FUNCTION_BLOCK FB_ObserverPattern_Test EXTENDS TcUnit.FB_TestSuite
// All observable types implements the same base methods for
// managing the list of observers, hence testing only one type
// of observable is enough. For instance, methods like, `Attach`,
// and `Detach`.
VAR
    fVal: LREAL;
END_VAR

TestAdd5CompatibleObserversExpectAll5();
TestAdd6IncompatibleObserversExpectNone();
TestAddDuplicateObserversExpectFailure();
TestAddMoreObserversThanAllowedExpectOnlyMaxCount();
TestCompatibleDataTypesExpectValuesToUpdate();
TestDataTypeConsistencyOfObservables();
TestDataTypeConsistencyOfObservers();
TestDetachAddedObserversExpectSuccess();
TestIncompatileDataTypesExpectNoValueChange();
TestObservableNotifyAlwaysUponWriteAccess();
TestObservableNotifyOnlyWhenValueChanged();
TestObservableNotifyUponAttachmentWithObservers();
TestObserverExternalWithCompatibleDataTypeExpectValueToUpdate();
TestOneObservableToManyObserversExpectAllToUpdateValueAccordingly();

METHOD PRIVATE TestAdd5CompatibleObserversExpectAll5
VAR_INST
    fbObservableReal: FB_Observable_REAL(TRUE);

    aObserverReal: ARRAY [1..5] OF FB_Observer_REAL;

    i: UDINT;
END_VAR
TcUnit.TEST('TestAdd5CompatibleObserversExpectAll5');

FOR i := 1 TO SIZEOF(aObserverReal)/SIZEOF(aObserverReal[1]) DO
    THIS^.AssertTrue(Condition := fbObservableReal.Attach(aObserverReal[i]),
                     Message := 'Failed to add compatible observer to observable');
END_FOR

THIS^.AssertEquals_UDINT(Expected := 5,
                         Actual := fbObservableReal.nObserverCount,
                         Message := 'Unexpected number of observers attached');

TcUnit.TEST_FINISHED();
END_METHOD

METHOD PRIVATE TestAdd6IncompatibleObserversExpectNone
VAR_INST
    // Test can be less manual with dynamic list
    fbObservableDint: FB_Observable_DINT(TRUE);
    fbObservableUdint: FB_Observable_UDINT(TRUE);
    fbObservableUint: FB_Observable_UINT(TRUE);
    fbObservableReal: FB_Observable_REAL(TRUE);
    fbObservableLreal: FB_Observable_LREAL(TRUE);

    fbObserverDint: ARRAY [1..6] OF FB_Observer_DINT;
    fbObserverUdint: ARRAY [1..6] OF FB_Observer_UDINT;
    fbObserverUint: ARRAY [1..6] OF FB_Observer_UINT;
    fbObserverLreal: ARRAY [1..6] OF FB_Observer_LREAL;
    fbObserverReal: ARRAY [1..6] OF FB_Observer_REAL;

    i: UDINT;
END_VAR
TcUnit.TEST('TestAdd6IncompatibleObserversExpectNone');

FOR i := 1 TO SIZEOF(fbObserverUdint)/SIZEOF(fbObserverUdint[1]) DO
    fbObservableDint.Attach(fbObserverUdint[i]);
    fbObservableDint.Attach(fbObserverUint[i]);
    fbObservableDint.Attach(fbObserverLreal[i]);
    fbObservableDint.Attach(fbObserverReal[i]);

    fbObservableUdint.Attach(fbObserverDint[i]);
    fbObservableUdint.Attach(fbObserverUint[i]);
    fbObservableUdint.Attach(fbObserverLreal[i]);
    fbObservableUdint.Attach(fbObserverReal[i]);

    fbObservableUint.Attach(fbObserverDint[i]);
    fbObservableUint.Attach(fbObserverUdint[i]);
    fbObservableUint.Attach(fbObserverLreal[i]);
    fbObservableUint.Attach(fbObserverReal[i]);

    fbObservableLreal.Attach(fbObserverDint[i]);
    fbObservableLreal.Attach(fbObserverUdint[i]);
    fbObservableLreal.Attach(fbObserverUint[i]);
    fbObservableLreal.Attach(fbObserverReal[i]);

    fbObservableReal.Attach(fbObserverDint[i]);
    fbObservableReal.Attach(fbObserverUdint[i]);
    fbObservableReal.Attach(fbObserverUint[i]);
    fbObservableReal.Attach(fbObserverLreal[i]);

END_FOR

THIS^.AssertEquals_UDINT(Expected := 0,
                         Actual := fbObservableDint.nObserverCount,
                         Message := 'Unexpected number of observers attached to observable type DINT');

THIS^.AssertEquals_UDINT(Expected := 0,
                         Actual := fbObservableUdint.nObserverCount,
                         Message := 'Unexpected number of observers attached to observable type UDINT');

THIS^.AssertEquals_UDINT(Expected := 0,
                         Actual := fbObservableUint.nObserverCount,
                         Message := 'Unexpected number of observers attached to observable type UINT');

THIS^.AssertEquals_UDINT(Expected := 0,
                         Actual := fbObservableLreal.nObserverCount,
                         Message := 'Unexpected number of observers attached to observable type LREAL');

THIS^.AssertEquals_UDINT(Expected := 0,
                         Actual := fbObservableReal.nObserverCount,
                         Message := 'Unexpected number of observers attached to observable type REAL');

TcUnit.TEST_FINISHED();
END_METHOD

METHOD PRIVATE TestAddDuplicateObserversExpectFailure
VAR_INST
    fbObservableReal: FB_Observable_REAL(TRUE);

    fbObserverReal: FB_Observer_REAL;

    i: UDINT;
END_VAR
TcUnit.TEST('TestAddDuplicateObserversExpectFailure');

FOR i := 1 TO 5 DO
    IF i = 1 THEN
        THIS^.AssertTrue(Condition := fbObservableReal.Attach(fbObserverReal),
                         Message := 'Failed to add compatible observer to observable');
    ELSE
        THIS^.AssertFalse(Condition := fbObservableReal.Attach(fbObserverReal),
                          Message := 'Observable should not add duplicate observers');
    END_IF
END_FOR

THIS^.AssertEquals_UDINT(Expected := 1,
                         Actual := fbObservableReal.nObserverCount,
                         Message := 'Unexpected number of observers attached');

TcUnit.TEST_FINISHED();
END_METHOD

METHOD PRIVATE TestAddMoreObserversThanAllowedExpectOnlyMaxCount
VAR_INST
    fbObservableReal: FB_Observable_REAL(TRUE);

    fbObserverReal: ARRAY [1..(TcBase.Param_Observer.cMaxNumberOfObservers+10)] OF FB_Observer_REAL;

    i: UDINT;
END_VAR
TcUnit.TEST('TestAddMoreObserversThanAllowedExpectOnlyMaxCount');

FOR i := 1 TO SIZEOF(fbObserverReal)/SIZEOF(fbObserverReal[1]) DO
    fbObservableReal.Attach(fbObserverReal[i]);
END_FOR

THIS^.AssertEquals_UDINT(Expected := TcBase.Param_Observer.cMaxNumberOfObservers,
                         Actual := fbObservableReal.nObserverCount,
                         Message := 'Unexpected number of observers attached');

TcUnit.TEST_FINISHED();
END_METHOD

METHOD PRIVATE TestCompatibleDataTypesExpectValuesToUpdate
VAR_INST
    fbObservableBool: FB_Observable_BOOL(TRUE);
    fbObservableByte: FB_Observable_BYTE(TRUE);
    fbObservableWord: FB_Observable_WORD(TRUE);
    fbObservableDword: FB_Observable_DWORD(TRUE);
    fbObservableLword: FB_Observable_LWORD(TRUE);
    fbObservableSint: FB_Observable_SINT(TRUE);
    fbObservableUsint: FB_Observable_USINT(TRUE);
    fbObservableInt: FB_Observable_INT(TRUE);
    fbObservableUint: FB_Observable_UINT(TRUE);
    fbObservableDint: FB_Observable_DINT(TRUE);
    fbObservableUdint: FB_Observable_UDINT(TRUE);
    fbObservableLint: FB_Observable_LINT(TRUE);
    fbObservableUlint: FB_Observable_ULINT(TRUE);
    fbObservableLreal: FB_Observable_LREAL(TRUE);
    fbObservableReal: FB_Observable_REAL(TRUE);

    fbObserverBool: FB_Observer_BOOL;
    fbObserverByte: FB_Observer_BYTE;
    fbObserverWord: FB_Observer_WORD;
    fbObserverDword: FB_Observer_DWORD;
    fbObserverLword: FB_Observer_LWORD;
    fbObserverSint: FB_Observer_SINT;
    fbObserverUsint: FB_Observer_USINT;
    fbObserverInt: FB_Observer_INT;
    fbObserverUint: FB_Observer_UINT;
    fbObserverDint: FB_Observer_DINT;
    fbObserverUdint: FB_Observer_UDINT;
    fbObserverLint: FB_Observer_LINT;
    fbObserverUlint: FB_Observer_ULINT;
    fbObserverLreal: FB_Observer_LREAL;
    fbObserverReal: FB_Observer_REAL;

    bVal: BOOL;
    i: UDINT;
END_VAR
TcUnit.TEST('TestCompatibleDataTypesExpectValuesToUpdate');

fbObservableBool.Attach(fbObserverBool);
fbObservableByte.Attach(fbObserverByte);
fbObservableWord.Attach(fbObserverWord);
fbObservableDword.Attach(fbObserverDword);
fbObservableLword.Attach(fbObserverLword);
fbObservableSint.Attach(fbObserverSint);
fbObservableUsint.Attach(fbObserverUsint);
fbObservableUint.Attach(fbObserverUint);
fbObservableInt.Attach(fbObserverInt);
fbObservableDint.Attach(fbObserverDint);
fbObservableUdint.Attach(fbObserverUdint);
fbObservableLint.Attach(fbObserverLint);
fbObservableUlint.Attach(fbObserverUlint);
fbObservableLreal.Attach(fbObserverLreal);
fbObservableReal.Attach(fbObserverReal);

FOR i := 1 TO 10 DO
    bVal := NOT bVal;
    fbObservableBool.bVal := bVal;
    fbObservableByte.nValue8 := TO_BYTE(i);
    fbObservableWord.nValue16 := TO_WORD(i);
    fbObservableDword.nValue32 := TO_DWORD(i);
    fbObservableLword.nValue64 := TO_LWORD(i);
    fbObservableSint.nValue8 := TO_SINT(i);
    fbObservableUsint.nValue8 := TO_USINT(i);
    fbObservableInt.nValue16 := TO_INT(i);
    fbObservableUint.nValue16 := TO_UINT(i);
    fbObservableDint.nValue32 := TO_DINT(i);
    fbObservableUdint.nValue32 := i;
    fbObservableLint.nValue64 := TO_LINT(i);
    fbObservableUlint.nValue64 := TO_ULINT(i);
    fbObservableLreal.fValue64 := TO_LREAL(i);
    fbObservableReal.fValue32 := TO_REAL(i);

    THIS^.AssertEquals_BOOL(Expected := bVal,
                            Actual := fbObserverBool.bValue,
                            Message := 'BOOL observer failed to update value according to observable');
    THIS^.AssertEquals_BYTE(Expected := TO_BYTE(i),
                            Actual := fbObserverByte.nValue8,
                            Message := 'BYTE observer failed to update value according to observable');
    THIS^.AssertEquals_WORD(Expected := TO_WORD(i),
                            Actual := fbObserverWord.nValue16,
                            Message := 'WORD observer failed to update value according to observable');
    THIS^.AssertEquals_DWORD(Expected := TO_DWORD(i),
                             Actual := fbObserverDword.nValue32,
                             Message := 'DWORD observer failed to update value according to observable');
    THIS^.AssertEquals_LWORD(Expected := TO_LWORD(i),
                             Actual := fbObserverLword.nValue64,
                             Message := 'LWORD observer failed to update value according to observable');
    THIS^.AssertEquals_SINT(Expected := TO_SINT(i),
                            Actual := fbObserverSint.nValue8,
                            Message := 'SINT observer failed to update value according to observable');
    THIS^.AssertEquals_USINT(Expected := TO_USINT(i),
                             Actual := fbObserverUsint.nValue8,
                             Message := 'USINT observer failed to update value according to observable');
    THIS^.AssertEquals_INT(Expected := TO_INT(i),
                           Actual := fbObserverInt.nValue16,
                           Message := 'INT observer failed to update value according to observable');
    THIS^.AssertEquals_UINT(Expected := TO_UINT(i),
                            Actual := fbObserverUint.nValue16,
                            Message := 'UINT observer failed to update value according to observable');
    THIS^.AssertEquals_DINT(Expected := TO_DINT(i),
                            Actual := fbObserverDint.nValue32,
                            Message := 'DINT observer failed to update value according to observable');
    THIS^.AssertEquals_UDINT(Expected := i,
                             Actual := fbObserverUdint.nValue32,
                             Message := 'UDINT observer failed to update value according to observable');
    THIS^.AssertEquals_LINT(Expected := TO_LINT(i),
                            Actual := fbObserverLint.nValue64,
                            Message := 'LINT observer failed to update value according to observable');
    THIS^.AssertEquals_LREAL(Expected := TO_LREAL(i),
                             Actual := fbObserverLreal.fValue64,
                             Delta := 0.01,
                             Message := 'LREAL observer failed to update value according to observable');
    THIS^.AssertEquals_REAL(Expected := TO_REAL(i),
                            Actual := fbObserverReal.fValue32,
                            Delta := 0.01,
                            Message := 'REAL observer failed to update value according to observable');
END_FOR

TcUnit.TEST_FINISHED();
END_METHOD

METHOD PRIVATE TestDataTypeConsistencyOfObservables
VAR_INST
    aTypes: ARRAY [1..15] OF __SYSTEM.TYPE_CLASS :=
        [
            __SYSTEM.TYPE_CLASS.TYPE_BOOL,
            __SYSTEM.TYPE_CLASS.TYPE_BYTE,
            __SYSTEM.TYPE_CLASS.TYPE_WORD,
            __SYSTEM.TYPE_CLASS.TYPE_DWORD,
            __SYSTEM.TYPE_CLASS.TYPE_LWORD,
            __SYSTEM.TYPE_CLASS.TYPE_SINT,
            __SYSTEM.TYPE_CLASS.TYPE_USINT,
            __SYSTEM.TYPE_CLASS.TYPE_INT,
            __SYSTEM.TYPE_CLASS.TYPE_UINT,
            __SYSTEM.TYPE_CLASS.TYPE_DINT,
            __SYSTEM.TYPE_CLASS.TYPE_UDINT,
            __SYSTEM.TYPE_CLASS.TYPE_LINT,
            __SYSTEM.TYPE_CLASS.TYPE_ULINT,
            __SYSTEM.TYPE_CLASS.TYPE_LREAL,
            __SYSTEM.TYPE_CLASS.TYPE_REAL
        ];

    fbList: FB_List;
    fbObservableBool: FB_Observable_BOOL(TRUE);
    fbObservableByte: FB_Observable_BYTE(TRUE);
    fbObservableWord: FB_Observable_WORD(TRUE);
    fbObservableDword: FB_Observable_DWORD(TRUE);
    fbObservableLword: FB_Observable_LWORD(TRUE);
    fbObservableSint: FB_Observable_SINT(TRUE);
    fbObservableUsint: FB_Observable_USINT(TRUE);
    fbObservableInt: FB_Observable_INT(TRUE);
    fbObservableUint: FB_Observable_UINT(TRUE);
    fbObservableDint: FB_Observable_DINT(TRUE);
    fbObservableUdint: FB_Observable_UDINT(TRUE);
    fbObservableLint: FB_Observable_LINT(TRUE);
    fbObservableUlint: FB_Observable_ULINT(TRUE);
    fbObservableLreal: FB_Observable_LREAL(TRUE);
    fbObservableReal: FB_Observable_REAL(TRUE);

    ipTmp: I_Observable;
    i: UDINT;
END_VAR
TcUnit.TEST('TestExpectConsistentDataTypeOfObservables');

fbList.AddItem(fbObservableBool);
fbList.AddItem(fbObservableByte);
fbList.AddItem(fbObservableWord);
fbList.AddItem(fbObservableDword);
fbList.AddItem(fbObservableLword);
fbList.AddItem(fbObservableSint);
fbList.AddItem(fbObservableUsint);
fbList.AddItem(fbObservableInt);
fbList.AddItem(fbObservableUint);
fbList.AddItem(fbObservableDint);
fbList.AddItem(fbObservableUdint);
fbList.AddItem(fbObservableLint);
fbList.AddItem(fbObservableUlint);
fbList.AddItem(fbObservableLreal);
fbList.AddItem(fbObservableReal);

FOR i := 1 TO SIZEOF(aTypes)/SIZEOF(aTypes[i]) DO
    __QUERYINTERFACE(fbList.ItemAt(TO_DINT(i - 1)), ipTmp);
    THIS^.AssertEquals_UDINT(Expected := aTypes[i],
                             Actual := ipTmp.nTypeClass,
                             Message := CONCAT('Inconsistent type class for observable tested at index ', TO_STRING(i)));
END_FOR

TcUnit.TEST_FINISHED();
END_METHOD

METHOD PRIVATE TestDataTypeConsistencyOfObservers
VAR_INST
    aTypes: ARRAY [1..15] OF __SYSTEM.TYPE_CLASS :=
        [
            __SYSTEM.TYPE_CLASS.TYPE_BOOL,
            __SYSTEM.TYPE_CLASS.TYPE_BYTE,
            __SYSTEM.TYPE_CLASS.TYPE_WORD,
            __SYSTEM.TYPE_CLASS.TYPE_DWORD,
            __SYSTEM.TYPE_CLASS.TYPE_LWORD,
            __SYSTEM.TYPE_CLASS.TYPE_SINT,
            __SYSTEM.TYPE_CLASS.TYPE_USINT,
            __SYSTEM.TYPE_CLASS.TYPE_INT,
            __SYSTEM.TYPE_CLASS.TYPE_UINT,
            __SYSTEM.TYPE_CLASS.TYPE_DINT,
            __SYSTEM.TYPE_CLASS.TYPE_UDINT,
            __SYSTEM.TYPE_CLASS.TYPE_LINT,
            __SYSTEM.TYPE_CLASS.TYPE_ULINT,
            __SYSTEM.TYPE_CLASS.TYPE_LREAL,
            __SYSTEM.TYPE_CLASS.TYPE_REAL
        ];

    fbList: FB_List;
    fbObserverBool: FB_Observer_BOOL;
    fbObserverByte: FB_Observer_BYTE;
    fbObserverWord: FB_Observer_WORD;
    fbObserverDword: FB_Observer_DWORD;
    fbObserverLword: FB_Observer_LWORD;
    fbObserverSint: FB_Observer_SINT;
    fbObserverUsint: FB_Observer_USINT;
    fbObserverInt: FB_Observer_INT;
    fbObserverUint: FB_Observer_UINT;
    fbObserverDint: FB_Observer_DINT;
    fbObserverUdint: FB_Observer_UDINT;
    fbObserverLint: FB_Observer_LINT;
    fbObserverUlint: FB_Observer_ULINT;
    fbObserverLreal: FB_Observer_LREAL;
    fbObserverReal: FB_Observer_REAL;

    ipTmp: I_Observer;
    i: UDINT;
END_VAR
TcUnit.TEST('TestExpectConsistentDataTypeOfObservers');

fbList.AddItem(fbObserverBool);
fbList.AddItem(fbObserverByte);
fbList.AddItem(fbObserverWord);
fbList.AddItem(fbObserverDword);
fbList.AddItem(fbObserverLword);
fbList.AddItem(fbObserverSint);
fbList.AddItem(fbObserverUsint);
fbList.AddItem(fbObserverInt);
fbList.AddItem(fbObserverUint);
fbList.AddItem(fbObserverDint);
fbList.AddItem(fbObserverUdint);
fbList.AddItem(fbObserverLint);
fbList.AddItem(fbObserverUlint);
fbList.AddItem(fbObserverLreal);
fbList.AddItem(fbObserverReal);

FOR i := 1 TO SIZEOF(aTypes)/SIZEOF(aTypes[i]) DO
    __QUERYINTERFACE(fbList.ItemAt(TO_DINT(i - 1)), ipTmp);
    THIS^.AssertEquals_UDINT(Expected := aTypes[i],
                             Actual := ipTmp.nTypeClass,
                             Message := CONCAT('Inconsistent type class for observable tested at index ', TO_STRING(i)));
END_FOR

TcUnit.TEST_FINISHED();
END_METHOD

METHOD PRIVATE TestDetachAddedObserversExpectSuccess
VAR_INST
    fbObservableReal: FB_Observable_REAL(TRUE);
    fbObserverReal: ARRAY [1..5] OF FB_Observer_REAL;

    i: UDINT;
END_VAR
TcUnit.TEST('TestDetachAddedObserversExpectSuccess');

FOR i := 1 TO SIZEOF(fbObserverReal)/SIZEOF(fbObserverReal[1]) DO
    fbObservableReal.Attach(fbObserverReal[i]);
END_FOR

FOR i := 1 TO SIZEOF(fbObserverReal)/SIZEOF(fbObserverReal[1]) DO
    THIS^.AssertTrue(Condition := fbObservableReal.Detach(fbObserverReal[i]),
                     Message := 'Failed to deatch added observer');

END_FOR

THIS^.AssertEquals_UDINT(Expected := 0,
                         Actual := fbObservableReal.nObserverCount,
                         Message := 'Unexpected number of observers attached');

TcUnit.TEST_FINISHED();
END_METHOD

METHOD PRIVATE TestIncompatileDataTypesExpectNoValueChange
VAR_INST
    fbObservableReal: FB_Observable_REAL(TRUE);

    fbObserverDint: FB_Observer_DINT;
    fbObserverUdint: FB_Observer_UDINT;
    fbObserverUint: FB_Observer_UINT;
    fbObserverLreal: FB_Observer_LREAL;

    i: UDINT;
END_VAR
TcUnit.TEST('TestIncompatileDataTypeObserverAndObservableExpectNoValueChange');

fbObservableReal.Attach(fbObserverDint);
fbObservableReal.Attach(fbObserverUdint);
fbObservableReal.Attach(fbObserverUint);
fbObservableReal.Attach(fbObserverLreal);

FOR i := 1 TO 10 DO
    fbObservableReal.fValue32 := TO_REAL(i);

    THIS^.AssertEquals_DINT(Expected := 0,
                            Actual := fbObserverDint.nValue32,
                            Message := 'DINT observer value is not 0, but it should be 0');

    THIS^.AssertEquals_UDINT(Expected := 0,
                            Actual := fbObserverUdint.nValue32,
                            Message := 'UDINT observer value is not 0, but it should be 0');

    THIS^.AssertEquals_UINT(Expected := 0,
                            Actual := fbObserverUint.nValue16,
                            Message := 'UINT observer value is not 0, but it should be 0');

    THIS^.AssertEquals_LREAL(Expected := 0,
                             Actual := fbObserverLreal.fValue64,
                             Delta := 0.001,
                             Message := 'LREAL observer value is not 0, but it should be 0');
END_FOR

TcUnit.TEST_FINISHED();
END_METHOD

METHOD PRIVATE TestObservableNotifyAlwaysUponWriteAccess
VAR_INST
    fbObservable: FB_Observable_LREAL(TRUE);
    fbObserver: FB_Observer_LREAL_;

    i: UDINT;
END_VAR
TcUnit.TEST('TestObservableNotifyAlwaysUponWriteAccess');

fbObservable.bNotifyWhenChanged := FALSE;
fbObservable.Attach(fbObserver);

// Expecte 1 update already because observable always update its observer upon
// attachment
THIS^.AssertEquals_UDINT(Expected := 1,
                         Actual := fbObserver.nUpdateCounter,
                         Message := 'Unexpected number of updates to observer');

FOR i := 1 TO 5 DO
    fbObservable.fValue64 := 1.0;
END_FOR

THIS^.AssertEquals_UDINT(Expected := 6,
                         Actual := fbObserver.nUpdateCounter,
                         Message := 'Unexpected number of updates to observer');

TcUnit.TEST_FINISHED();
END_METHOD

METHOD PRIVATE TestObservableNotifyOnlyWhenValueChanged
VAR_INST
    fbObservable: FB_Observable_LREAL(TRUE);
    fbObserver: FB_Observer_LREAL_;
    aVal: ARRAY [1..5] OF LREAL :=
        [2.7183, 3.1415, -1, 1.6180, 6.6261];

    i: UDINT;
    j: UDINT;
END_VAR
TcUnit.TEST('TestObservableNotifyOnlyWhenValueChanged');

fbObservable.Attach(fbObserver);

// Expect 1 update already because observable always update its observer upon
// attachment
THIS^.AssertEquals_UDINT(Expected := 1,
                         Actual := fbObserver.nUpdateCounter,
                         Message := 'Unexpected number of updates to observer');

FOR i := 1 TO SIZEOF(aVal)/SIZEOF(aVal[1]) DO
    FOR j := 1 TO 5 DO
        fbObservable.fValue64 := aVal[i];
    END_FOR

    THIS^.AssertEquals_UDINT(Expected := i + 1,
                             Actual := fbObserver.nUpdateCounter,
                             Message := 'Unexpected number of updates to observer');
END_FOR


TcUnit.TEST_FINISHED();
END_METHOD

METHOD PRIVATE TestObservableNotifyUponAttachmentWithObservers
VAR_INST
    fbObservable: FB_Observable_LREAL(TRUE);
    aObserver: ARRAY [1..5] OF FB_Observer_LREAL_;

    i: UDINT;
END_VAR
TcUnit.TEST('TestObservableNotifyUponAttachmentWithObservers');

fbObservable.fValue64 := 100.0;

FOR i := 1 TO SIZEOF(aObserver)/SIZEOF(aObserver[1]) DO
    fbObservable.Attach(aObserver[i]);
END_FOR

FOR i := 1 TO SIZEOF(aObserver)/SIZEOF(aObserver[1]) DO
    THIS^.AssertEquals_LREAL(Expected := fbObservable.fValue64,
                             Actual := aObserver[i].fValue64,
                             Delta := 0.01,
                             Message := 'Observer$'s value is not matching its observable upon attachment');
    THIS^.AssertEquals_UDINT(Expected := 1,
                             Actual := aObserver[i].nUpdateCounter,
                             Message := 'Unexpected number of updates to observer');
END_FOR

TcUnit.TEST_FINISHED();
END_METHOD

METHOD PRIVATE TestObserverExternalWithCompatibleDataTypeExpectValueToUpdate
VAR_INST
    fbObservableLreal: FB_Observable_LREAL(TRUE);
    fbObserverExt: FB_ObserverExt(THIS^.fVal);
    aTestVal: ARRAY [1..5] OF LREAL :=
        [2.7183, 3.1415, -1, 1.6180, 6.6261];
    i: UDINT;
END_VAR
TcUnit.TEST('TestObserverExternalWithCompatibleDataTypeExpectValueToUpdate');

fbObservableLreal.Attach(fbObserverExt);

FOR i := 1 TO SIZEOF(aTestVal)/SIZEOF(aTestVal[1]) DO
    fbObservableLreal.fValue64 := aTestVal[i];
    THIS^.AssertEquals_LREAL(Expected := aTestVal[i],
                             Actual := THIS^.fVal,
                             Delta := 0.001,
                             Message := 'External observer typed LREAL failed to update value according to observable');
END_FOR

TcUnit.TEST_FINISHED();
END_METHOD

METHOD PRIVATE TestOneObservableToManyObserversExpectAllToUpdateValueAccordingly
VAR_INST
    fbObservableLreal: FB_Observable_LREAL(TRUE);
    aObservers: ARRAY [1..5] OF FB_Observer_LREAL;
    aTestVal: ARRAY [1..5] OF LREAL :=
        [2.7183, 3.1415, -1, 1.6180, 6.6261];
    i: UDINT;
    j: UDINT;
END_VAR
TcUnit.TEST('TestOneObservableToManyObserversExpectAllToUpdateValueAccordingly');

FOR i := 1 TO SIZEOF(aObservers)/SIZEOF(aObservers[1]) DO
    fbObservableLreal.Attach(aObservers[i]);
END_FOR

FOR i := 1 TO SIZEOF(aTestVal)/SIZEOF(aTestVal[1]) DO
    fbObservableLreal.fValue64 := aTestVal[i];
    FOR j := 1 TO SIZEOF(aObservers)/SIZEOF(aObservers[1]) DO
        THIS^.AssertEquals_LREAL(Expected := aTestVal[i],
                         Actual := aObservers[j].fValue64,
                         Delta := 0.001,
                         Message := ' typed LREAL failed to update value according to observable');
    END_FOR
END_FOR

TcUnit.TEST_FINISHED();
END_METHOD

END_FUNCTION_BLOCK

(* stored: Version 1.1.0.1, ProductVersion 3.1.4024.12
   POU FB_ObserverPattern_Test: Id {9669889e-5dc1-4a5e-b021-9809da0da496}, SpecialFunc None
   Method TestAdd5CompatibleObserversExpectAll5: Id {791da87e-3b1e-4df9-be32-6b1c00308983}
   Method TestAdd6IncompatibleObserversExpectNone: Id {f008ceac-1587-4d6c-8c53-a475f778f5b0}
   Method TestAddDuplicateObserversExpectFailure: Id {541af2f9-185f-04a2-08d3-89d5044bece3}
   Method TestAddMoreObserversThanAllowedExpectOnlyMaxCount: Id {0c149026-c1e8-4c39-92b6-923e4107cb0e}
   Method TestCompatibleDataTypesExpectValuesToUpdate: Id {a0c42179-d282-4d90-9f50-7c032bf816e4}
   Method TestDataTypeConsistencyOfObservables: Id {b35d1778-9728-4d09-b056-cd7e607ea8b6}
   Method TestDataTypeConsistencyOfObservers: Id {52e78a6a-e28a-49fb-b8c1-34fea3e87f66}
   Method TestDetachAddedObserversExpectSuccess: Id {d0a8dd44-ed9b-0741-3658-2e78db7d42e9}
   Method TestIncompatileDataTypesExpectNoValueChange: Id {0979a056-7376-4db3-99e3-658aa0013606}
   Method TestObservableNotifyAlwaysUponWriteAccess: Id {6bd03110-3809-4b9a-be1d-26037011bd0e}
   Method TestObservableNotifyOnlyWhenValueChanged: Id {22acf0a5-0c89-4f61-b880-4714e2c4dc93}
   Method TestObservableNotifyUponAttachmentWithObservers: Id {80e2d94c-c26a-4a53-990f-cd6227123e7b}
   Method TestObserverExternalWithCompatibleDataTypeExpectValueToUpdate: Id {10be65a2-219d-0b3c-1bbe-50f6d1861ef6}
   Method TestOneObservableToManyObserversExpectAllToUpdateValueAccordingly: Id {6c79a3a7-11b6-0c82-0376-6a2fc2c49511} *)
